FUNCTION angAxis2Rot : Mat3d
VAR_INPUT
	i_angle :LREAL;
	i_axis :Vec3d;
END_VAR
VAR
	cAng, sAng :LREAL;
	rx,ry,rz :LREAL;
END_VAR

IF norm(i_axis)<g_smallNum THEN
	angAxis2Rot := g_eye3d;
	RETURN;
END_IF

cAng :=COS(i_angle);
sAng := SIN(i_angle);
rx:=i_axis[1];
ry:=i_axis[2];
rz:=i_axis[3];

angAxis2Rot[1,1]:=rx*rx*(1-cAng)+cAng;
angAxis2Rot[2,1]:=rx*ry*(1-cAng)+rz*sAng;
angAxis2Rot[3,1]:=rx*rz*(1-cAng)-ry*sAng;

angAxis2Rot[1,2]:=rx*ry*(1-cAng)-rz*sAng;
angAxis2Rot[2,2]:=ry*ry*(1-cAng)+cAng;
angAxis2Rot[3,2]:=ry*rz*(1-cAng)+rx*sAng;

angAxis2Rot[1,3]:=rx*rz*(1-cAng)+ry*sAng;
angAxis2Rot[2,3]:=ry*rz*(1-cAng)-rx*sAng;
angAxis2Rot[3,3]:=rz*rz*(1-cAng)+cAng;

END_FUNCTION

(* stored: Version 1.1.0.1, ProductVersion 3.1.4024.11
   POU angAxis2Rot: Id {e5ebf543-ca8b-4cbd-9a97-b6a387ef41b1}, SpecialFunc None *)
